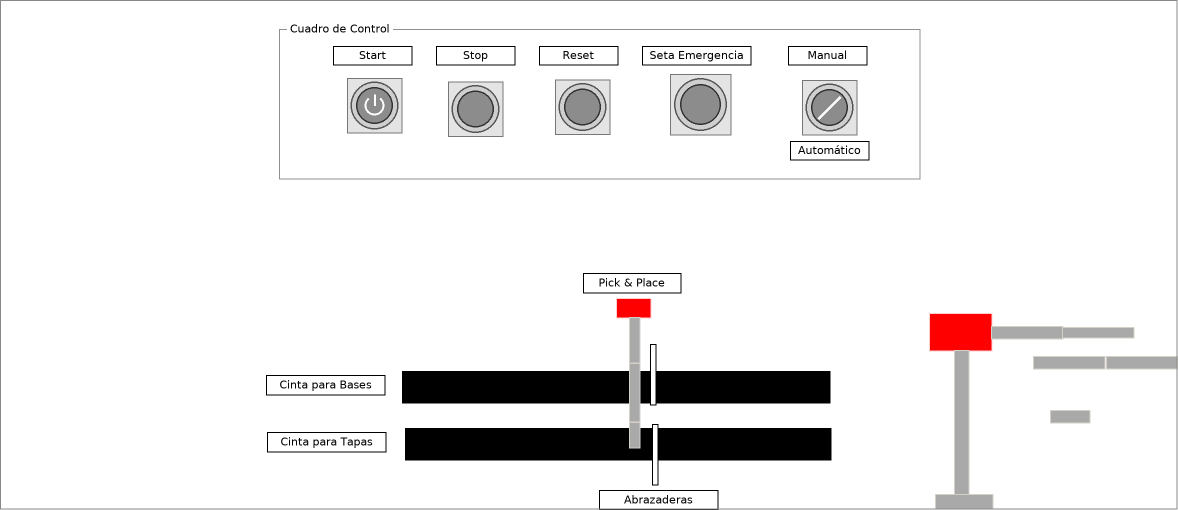
VISUALIZATION HMI  // 1178x510
    GroupBox (279,21 641x158), "Cuadro de Control"
        PowerSwitch (64,57 63x55), variable: GVLvars.botonStart, behaviour: TOGGLE, style: Switch-PowerSwitch-Gray
        PushSwitch (169,58 55x60), variable: GVLvars.botonStop, behaviour: TOGGLE, style: Switch-PushSwitch-Gray
        PushSwitch (276,56 55x60), variable: GVLvars.botonReset, behaviour: TOGGLE, style: Switch-PushSwitch-Gray
        PushSwitchLed (390,53 63x61), variable: GVLvars.seta, behaviour: TOGGLE, style: Switch-PushSwitchLed-Gray
        Rectangle (54,25 79x19), "Start"
        Rectangle (157,25 79x19), "Stop"
        Rectangle (260,25 79x19), "Reset"
        Rectangle (363,25 109x19), "Seta Emergencia"
        Rectangle (509,25 79x19), "Manual"
        Rectangle (511,120 79x19), "Automático"
        RotarySwitch (523,59 55x55), variable: GVLvars.modoManual, behaviour: TOGGLE, style: Switch-RotarySwitch-Gray
    Rectangle (405,428 426x32), colour toggle: GVLvars.cintaBases
        toggle GVLvars.cintaBases
    Rectangle (402,371 428x32), colour toggle: GVLvars.cintaTapas
        toggle GVLvars.cintaTapas
    Rectangle (616,298 35x20)
    Rectangle (629,317 11x46)
    Rectangle (629,363 11x59), colour toggle: GVLvars.PickPlace_MoverX, invisible if: NOT GVLvars.PickPlace_MoverX
        toggle GVLvars.PickPlace_MoverX
    Rectangle (629,422 11x26), colour toggle: GVLvars.PickPlace_MoverX, invisible if: NOT GVLvars.PickPlace_MoverX
        toggle GVLvars.PickPlace_MoverX
    Rectangle (583,273 98x20), "Pick & Place"
    Rectangle (929,313 63x38)
    Rectangle (954,350 15x145)
    Rectangle (991,326 72x13)
    Rectangle (1062,327 72x11), colour toggle: GVLvars.PickPlace_MoverX, invisible if: NOT GVLvars.PickPlace_MoverX
        toggle GVLvars.PickPlace_MoverX
    Rectangle (1106,356 72x13), angle 89, colour toggle: MAIN.bajarSinObjeto, invisible if: NOT MAIN.bajarSinObjeto
        toggle MAIN.bajarSinObjeto
    Rectangle (1033,356 72x13), angle 89, invisible if: NOT MAIN.bajarConObjeto
    Rectangle (1050,410 40x13), angle 89, colour toggle: MAIN.bajarConObjeto, invisible if: NOT MAIN.bajarConObjeto
        toggle MAIN.bajarConObjeto
    Rectangle (623,371 61x6), angle 90, colour toggle: GVLvars.cerrarAbrazaderaTapa
        toggle GVLvars.cerrarAbrazaderaTapa
    Rectangle (625,451 61x6), angle 90, colour toggle: GVLvars.cerrarAbrazaderaBase
        toggle GVLvars.cerrarAbrazaderaBase
    Rectangle (266,375 119x20), "Cinta para Bases"
    Rectangle (267,432 119x20), "Cinta para Tapas"
    Rectangle (599,490 119x20), "Abrazaderas"
    Rectangle (935,494 58x15)
END_VISUALIZATION

(* stored: Version 1.1.0.1, ProductVersion 3.1.4024.15
   Visu HMI: Id {2b889e45-c01f-4872-85cb-6ebc6dea87a9} *)
